// Mitsubishi GX Works2 project: Modbus TCP   PLC: Q03UDV

PROGRAM MAIN
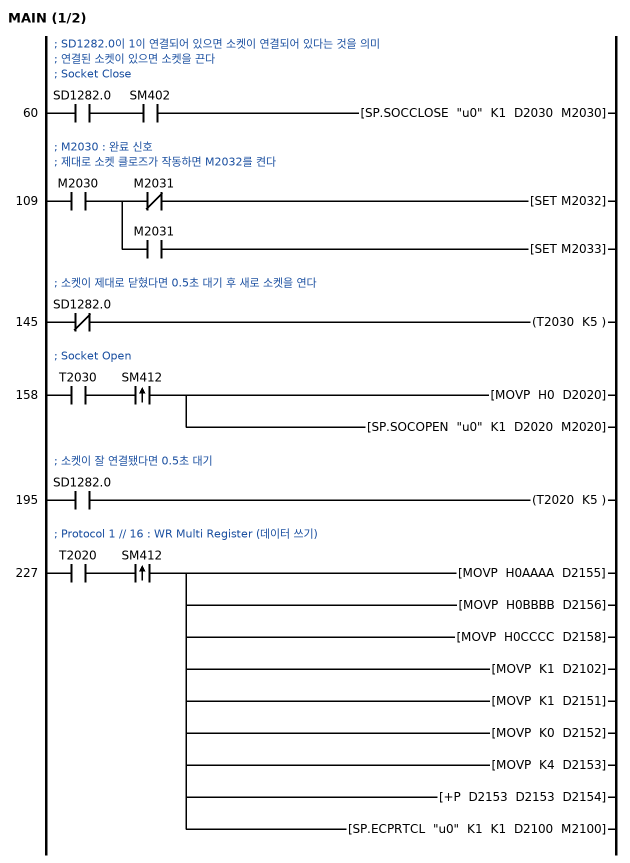
; SD1282.0이 1이 연결되어 있으면 소켓이 연결되어 있다는 것을 의미
; 연결된 소켓이 있으면 소켓을 끈다
; Socket Close
60    LD      SD1282.0
      AND     SM402
      SP.SOCCLOSE "u0" K1 D2030 M2030
; M2030 : 완료 신호
; 제대로 소켓 클로즈가 작동하면 M2032를 켠다
109   LD      M2030
      MPS
      ANI     M2031
      SET     M2032
      MPP
      AND     M2031
      SET     M2033
; 소켓이 제대로 닫혔다면 0.5초 대기 후 새로 소켓을 연다
145   LDI     SD1282.0
      OUT     T2030 K5
; Socket Open
158   LD      T2030
      ANDP    SM412
      MOVP    H0 D2020
      SP.SOCOPEN "u0" K1 D2020 M2020
; 소켓이 잘 연결됐다면 0.5초 대기
195   LD      SD1282.0
      OUT     T2020 K5
; Protocol 1 // 16 : WR Multi Register (데이터 쓰기)
227   LD      T2020
      ANDP    SM412
      MOVP    H0AAAA D2155
      MOVP    H0BBBB D2156
      MOVP    H0CCCC D2158
      MOVP    K1 D2102
      MOVP    K1 D2151
      MOVP    K0 D2152
      MOVP    K4 D2153
      +P      D2153 D2153 D2154
      SP.ECPRTCL "u0" K1 K1 D2100 M2100
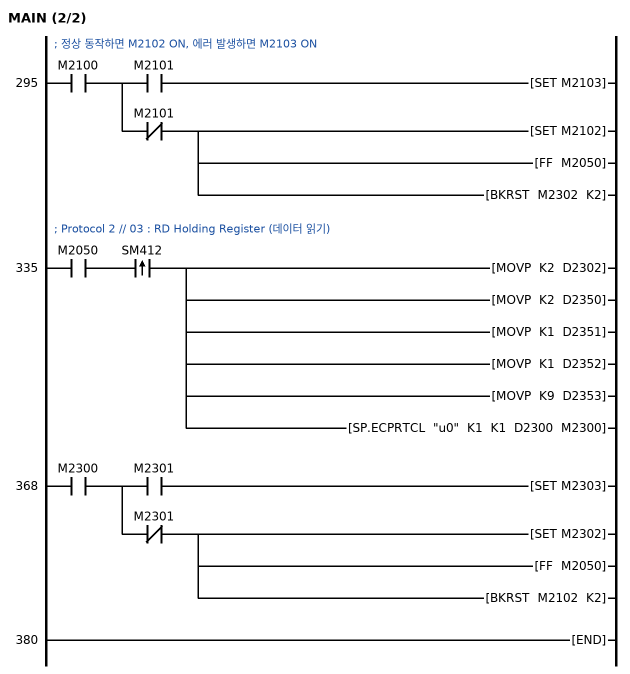
; 정상 동작하면 M2102 ON, 에러 발생하면 M2103 ON
295   LD      M2100
      MPS
      AND     M2101
      SET     M2103
      MPP
      ANI     M2101
      SET     M2102
      FF      M2050
      BKRST   M2302 K2
; Protocol 2 // 03 : RD Holding Register (데이터 읽기)
335   LD      M2050
      ANDP    SM412
      MOVP    K2 D2302
      MOVP    K2 D2350
      MOVP    K1 D2351
      MOVP    K1 D2352
      MOVP    K9 D2353
      SP.ECPRTCL "u0" K1 K1 D2300 M2300
368   LD      M2300
      MPS
      AND     M2301
      SET     M2303
      MPP
      ANI     M2301
      SET     M2302
      FF      M2050
      BKRST   M2102 K2
380   END
END_PROGRAM
